TYPE ST_System_HOWW_Parameter :
STRUCT
	AutoQuittierung			: BOOL;
END_STRUCT
END_TYPE

(* stored: Version 1.1.0.1, ProductVersion 3.1.4024.9
   DUT ST_System_HOWW_Parameter: Id {09f00f2d-c081-4f47-8b04-385b1090d967} *)
